// TwinCAT 3 PLC project TXI_SAT
// Title: mr3k3-mr4k3-mr2l1-mr3l1-sat
// Company: SLAC
// ProjectVersion: 0.0.0
// ProgramVersion: 3.1.4022.7
// libraries:
//   lcls-twincat-motion, * (SLAC)
//   Tc2_EtherCAT, * (Beckhoff Automation GmbH)
//   Tc2_Standard, * (Beckhoff Automation GmbH)
//   Tc2_System, * (Beckhoff Automation GmbH)
//   Tc3_Module, * (Beckhoff Automation GmbH)
// project tree:
//   / PlcTask.TcTTO
//   POUs/ MAIN.TcPOU
// real-time tasks:
//   TASK PlcTask: cycle T#10ms, priority 20, ADS port 350
// motion (NC):
//   TASK NC-Task 1 SAF: cycle T#2ms, priority 4, ADS port 501
//   TASK NC-Task 1 SVB: cycle T#10ms, priority 8, ADS port 511
//   AXIS M3K3 X (id 1)
//     Dynamic: AccelerationMaximum=100, DecelerationMaximum=100, Acceleration=100, Deceleration=100, DelayTime=0.008
//     Velo: Maximum=0.4
//     OtherSettings: AllowMotionCmdToSlave=true
//     encoder EncType=29
//       EncPara: ScaleFactorNumerator=5e-06, MaxCount=#xffffffff
//         Inc: RefSoftSyncMask=#x0000ffff
//     drive DrvType=24
//       DrvPara: Inverse=true
//         Analog: VeloReferenz=20, ScaleFactorActTorque=0.1
//         TimeComp: TaskDelayCycles=1
//     controller CtrType=2
//       CtrPara: PriorControlFactor=1
//         PosDiffControl: Range=0.3
//         PID: DeadBandPosition=0.1
//         Observer: BandWidth=20
//   AXIS M3K3 Y (id 2)
//     Dynamic: AccelerationMaximum=100, DecelerationMaximum=100, Acceleration=100, Deceleration=100, DelayTime=0.008
//     Velo: Maximum=0.3
//     OtherSettings: AllowMotionCmdToSlave=true
//     encoder EncType=29
//       EncPara: ScaleFactorNumerator=5e-06, MaxCount=#xffffffff
//         Inc: RefSoftSyncMask=#x0000ffff
//     drive DrvType=24
//       DrvPara: Inverse=true
//         Analog: VeloReferenz=1.25, ScaleFactorActTorque=0.1
//         TimeComp: TaskDelayCycles=1
//     controller CtrType=2
//       CtrPara: PriorControlFactor=1
//         PosDiffControl: Range=0.3
//         PID: DeadBandPosition=0.1
//         Observer: BandWidth=20
//   AXIS M3K3 rX (id 3)
//     General: UnitName=urad
//     Dynamic: AccelerationMaximum=100, DecelerationMaximum=100, Acceleration=100, Deceleration=100, DelayTime=0.008
//     Velo: Maximum=35
//     OtherSettings: AllowMotionCmdToSlave=true
//     encoder EncType=29
//       EncPara: ScaleFactorNumerator=0.001796, MaxCount=#xffffffff
//         Inc: RefSoftSyncMask=#x0000ffff
//     drive DrvType=24
//       Analog: VeloReferenz=87.7, ScaleFactorActTorque=0.1
//       TimeComp: TaskDelayCycles=1
//     controller CtrType=2
//       CtrPara: PriorControlFactor=1
//         PosDiffControl: Range=10
//         PID: DeadBandPosition=10
//         Observer: BandWidth=20
//   AXIS M4K3 X (id 4)
//     Dynamic: AccelerationMaximum=100, DecelerationMaximum=100, Acceleration=100, Deceleration=100, DelayTime=0.008
//     Velo: Maximum=0.3
//     OtherSettings: AllowMotionCmdToSlave=true
//     encoder EncType=29
//       EncPara: ScaleFactorNumerator=5e-06, MaxCount=#xffffffff
//         Inc: RefSoftSyncMask=#x0000ffff
//     drive DrvType=24
//       Analog: VeloReferenz=20, ScaleFactorActTorque=0.1
//       TimeComp: TaskDelayCycles=1
//     controller CtrType=2
//       CtrPara: PriorControlFactor=1
//         PosDiffControl: Range=0.3
//         PID: DeadBandPosition=0.1
//         Observer: BandWidth=20
//   AXIS M4K3 Y (id 5)
//     Dynamic: AccelerationMaximum=100, DecelerationMaximum=100, Acceleration=100, Deceleration=100, DelayTime=0.008
//     Velo: Maximum=0.3
//     OtherSettings: AllowMotionCmdToSlave=true
//     encoder EncType=29
//       EncPara: ScaleFactorNumerator=5e-06, MaxCount=#xffffffff
//         Inc: RefSoftSyncMask=#x0000ffff
//     drive DrvType=24
//       DrvPara: Inverse=true
//         Analog: VeloReferenz=1.25, ScaleFactorActTorque=0.1
//         TimeComp: TaskDelayCycles=1
//     controller CtrType=2
//       CtrPara: PriorControlFactor=1
//         PosDiffControl: Range=0.3
//         PID: DeadBandPosition=1
//         Observer: BandWidth=20
//   AXIS M4K3 rY (id 6)
//     General: UnitName=urad
//     Dynamic: AccelerationMaximum=100, DecelerationMaximum=100, Acceleration=100, Deceleration=100, DelayTime=0.008
//     Velo: Maximum=35
//     OtherSettings: AllowMotionCmdToSlave=true
//     encoder EncType=29
//       EncPara: ScaleFactorNumerator=0.0025316, MaxCount=#xffffffff
//         Inc: RefSoftSyncMask=#x0000ffff
//     drive DrvType=24
//       Analog: VeloReferenz=125, ScaleFactorActTorque=0.1
//       TimeComp: TaskDelayCycles=1
//     controller CtrType=2
//       CtrPara: PriorControlFactor=1
//         PosDiffControl: Range=10
//         PID: DeadBandPosition=0.1
//         Observer: BandWidth=20
//   AXIS M2L1 X (id 7)
//     Dynamic: AccelerationMaximum=100, DecelerationMaximum=100, Acceleration=100, Deceleration=100, DelayTime=0.008
//     Velo: Maximum=0.4
//     OtherSettings: AllowMotionCmdToSlave=true
//     encoder EncType=29
//       EncPara: ScaleFactorNumerator=5e-06, MaxCount=#xffffffff
//         Inc: RefSoftSyncMask=#x0000ffff
//     drive DrvType=24
//       DrvPara: Inverse=true
//         Analog: VeloReferenz=20, ScaleFactorActTorque=0.1
//         TimeComp: TaskDelayCycles=1
//     controller CtrType=2
//       CtrPara: PriorControlFactor=1
//         PosDiffControl: Range=0.3
//         PID: DeadBandPosition=0.1
//         Observer: BandWidth=20
//   AXIS M2L1 Y (id 8)
//     Dynamic: AccelerationMaximum=100, DecelerationMaximum=100, Acceleration=100, Deceleration=100, DelayTime=0.008
//     Velo: Maximum=0.3
//     OtherSettings: AllowMotionCmdToSlave=true
//     encoder EncType=29
//       EncPara: ScaleFactorNumerator=5e-06, MaxCount=#xffffffff
//         Inc: RefSoftSyncMask=#x0000ffff
//     drive DrvType=24
//       DrvPara: Inverse=true
//         Analog: VeloReferenz=1.25, ScaleFactorActTorque=0.1
//         TimeComp: TaskDelayCycles=1
//     controller CtrType=2
//       CtrPara: PriorControlFactor=1
//         PosDiffControl: Range=0.3
//         PID: DeadBandPosition=0.1
//         Observer: BandWidth=20
//   AXIS M2L1 rX (id 9)
//     General: UnitName=urad
//     Dynamic: AccelerationMaximum=100, DecelerationMaximum=100, Acceleration=100, Deceleration=100, DelayTime=0.008
//     Velo: Maximum=35
//     OtherSettings: AllowMotionCmdToSlave=true
//     encoder EncType=29
//       EncPara: ScaleFactorNumerator=0.001796, MaxCount=#xffffffff
//         Inc: RefSoftSyncMask=#x0000ffff
//     drive DrvType=24
//       Analog: VeloReferenz=87.7, ScaleFactorActTorque=0.1
//       TimeComp: TaskDelayCycles=1
//     controller CtrType=2
//       CtrPara: PriorControlFactor=1
//         PosDiffControl: Range=10
//         PID: DeadBandPosition=10
//         Observer: BandWidth=20
//   AXIS M3L1 X (id 10)
//     Dynamic: AccelerationMaximum=100, DecelerationMaximum=100, Acceleration=100, Deceleration=100, DelayTime=0.008
//     Velo: Maximum=0.3
//     OtherSettings: AllowMotionCmdToSlave=true
//     encoder EncType=29
//       EncPara: ScaleFactorNumerator=5e-06, MaxCount=#xffffffff
//         Inc: RefSoftSyncMask=#x0000ffff
//     drive DrvType=24
//       DrvPara: Inverse=true
//         Analog: VeloReferenz=20, ScaleFactorActTorque=0.1
//         TimeComp: TaskDelayCycles=1
//     controller CtrType=2
//       CtrPara: PriorControlFactor=1
//         PosDiffControl: Range=0.3
//         PID: DeadBandPosition=0.1
//         Observer: BandWidth=20
//   AXIS M3L1 Y (id 11)
//     Dynamic: AccelerationMaximum=100, DecelerationMaximum=100, Acceleration=100, Deceleration=100, DelayTime=0.008
//     Velo: Maximum=0.35
//     OtherSettings: AllowMotionCmdToSlave=true
//     encoder EncType=29
//       EncPara: ScaleFactorNumerator=5e-06, MaxCount=#xffffffff
//         Inc: RefSoftSyncMask=#x0000ffff
//     drive DrvType=24
//       DrvPara: Inverse=true
//         Analog: VeloReferenz=1.25, ScaleFactorActTorque=0.1
//         TimeComp: TaskDelayCycles=1
//     controller CtrType=2
//       CtrPara: PriorControlFactor=1
//         PosDiffControl: Range=0.3
//         PID: DeadBandPosition=1
//         Observer: BandWidth=20
//   AXIS M3L1 rY (id 12)
//     General: UnitName=urad
//     Dynamic: AccelerationMaximum=100, DecelerationMaximum=100, Acceleration=100, Deceleration=100, DelayTime=0.008
//     Velo: Maximum=35
//     OtherSettings: AllowMotionCmdToSlave=true
//     encoder EncType=29
//       EncPara: ScaleFactorNumerator=0.0025316, MaxCount=#xffffffff
//         Inc: RefSoftSyncMask=#x0000ffff
//     drive DrvType=24
//       Analog: VeloReferenz=125, ScaleFactorActTorque=0.1
//       TimeComp: TaskDelayCycles=1
//     controller CtrType=2
//       CtrPara: PriorControlFactor=1
//         PosDiffControl: Range=10
//         PID: PosExtKp=15, DeadBandPosition=0.1
//         Observer: BandWidth=20
//   AXIS MMS-BEND (id 13)
//     Dynamic: AccelerationMaximum=0.6, DecelerationMaximum=0.6, Acceleration=0.6, Deceleration=0.6, Jerk=1.2, DelayTime=0.008
//     Velo: Maximum=0.05
//     OtherSettings: AllowMotionCmdToSlave=true
//     encoder EncType=29
//       EncPara: ScaleFactorNumerator=1e-06, MaxCount=#xffffffff
//         SoftEndMinControl: Range=6.4549
//         SoftEndMaxControl: Range=16.0941
//         Inc: RefSoftSyncMask=#x0000ffff
//     drive DrvType=24
//       DrvPara: Inverse=true
//         Analog: VeloReferenz=0.1, ScaleFactorActTorque=0.1
//         TimeComp: TaskDelayCycles=1
//     controller CtrType=2
//       CtrPara: PriorControlFactor=1
//         PosDiffControl: Range=0.2
//         PID: PosKp=15, PosExtKp=1, DeadBandPosition=0.001
//         Observer: BandWidth=20
// I/O:
//   DEVICE Device 1 (EtherCAT), AmsNetId 172.21.84.181.2.1
//     Term 1 (EK1200) [EK1200-5000 EtherCAT Power supply (2A E-Bus)]
//       Term 24 (EL3052) [EL3052 2Ch. Ana. Input 4-20mA]
//       Term 25 (EL3202-0010) [EL3202-0010 2Ch. Ana. Input PT100 (RTD), High Precision]
//       Term 26 (EL7031) [EL7031 1Ch. Stepper motor output stage (24V, 1.5A)]
//       Term 2 (EK1122) [EK1122 2 port EtherCAT junction]
//         TXI K (EK1100) [EK1100 EtherCAT Coupler (2A E-Bus)]
//           M3K3 XY (EL5042)
//           M3K3 rX M4K3 X (EL5042)
//           M4K3 YrY (EL5042)
//           Term 7 (EL9221-5000) [EL9221-5000 Overcurrent protection 24V DC, 1Ch., max. 10A, adjustable]
//           M3K3 X (EL7041-0052)
//           M3K3 Y  (EL7041-0052)
//           M3K3 rX (EL7041-0052)
//           Term 11 (EL9221-5000)
//           M4K3 X (EL7041-0052)
//           M4K3 Y (EL7041-0052) [EL7041-0052 1Ch. Stepper motor output stage (50V, 5A)]
//           M4K3 rY (EL7041-0052) [EL7041-0052 1Ch. Stepper motor output stage (50V, 5A)]
//           Term 15 (EL9410) [EL9410 E-Bus Power Supplier  (Diagnostics)]
//           Term 16 (EL1004)
//           Term 17 (EL3204)
//           Term 18 (EL3204)
//           Term 19 (EL3202-0010)
//           Term 20 (EL3202-0010)
//           Term 21 (EL3054)
//           Term 97 (EL9011)
//         Term 22 (EK1100) [EK1100 EtherCAT Coupler (2A E-Bus)]
//           EL7041_MMS_BEND
//           EL5042_MMS_BEND [EL5042 2Ch. BiSS-C Encoder]
//           EL3202-0010_MMS_BEND [EL3202-0010 2Ch. Ana. Input PT100 (RTD), High Precision]
//           EL3202-0010_MMS_BEND_2 [EL3202-0010 2Ch. Ana. Input PT100 (RTD), High Precision]
//           Term 30 (EL9011)
//         TXI L (EK1100) [EK1100 EtherCAT Coupler (2A E-Bus)]
//           M2L1 XY (EL5042)
//           M2L1 rX M3L1 X (EL5042)
//           M3L1 YrY(EL5042)
//           Term 48 (EL9221-5000)
//           M2L1 X (EL7041-0052) [EL7041-0052 1Ch. Stepper motor output stage (50V, 5A)]
//           M2L1 Y (EL7041-0052) [EL7041-0052 1Ch. Stepper motor output stage (50V, 5A)]
//           M2L1 rX (EL7041-0052) [EL7041-0052 1Ch. Stepper motor output stage (50V, 5A)]
//           Term 52 (EL9221-5000)
//           M3L1 X (EL7041-0052) [EL7041-0052 1Ch. Stepper motor output stage (50V, 5A)]
//           M3L1 Y (EL7041-0052)
//           M3L1 rY (EL7041-0052) [EL7041-0052 1Ch. Stepper motor output stage (50V, 5A)]
//           Term 56 (EL9410)
//           Term 57 (EL3204)
//           Term 58 (EL3204)
//           Term 59 (EL3202-0010)
//           Term 60 (EL3202-0010)
//           Term 61 (EL3054) [EL3054 4Ch. Ana. Input 4-20mA]
//           Term 63 (EL9011)
// variable links:
//   (this object) <-> Device 1 (EtherCAT)/Term 1 (EK1200)/Term 2 (EK1122)/TXI K (EK1100)/M3K3 X (EL7041-0052)
//     Drive/Inputs/In/nState1 @bit 3 <-> STM Status/Status/Error
//     Drive/Inputs/In/nState1 @bit 5 <-> STM Status/Status/Moving negative
//     Drive/Inputs/In/nState1 @bit 4 <-> STM Status/Status/Moving positive
//     Drive/Inputs/In/nState1 @bit 1 <-> STM Status/Status/Ready
//     Drive/Inputs/In/nState1 <-> STM Status/Status/Ready to enable
//     Drive/Inputs/In/nState1 @bit 6 <-> STM Status/Status/Torque reduced
//     Drive/Inputs/In/nState1 @bit 2 <-> STM Status/Status/Warning
//     Drive/Inputs/In/nState2 @bit 3 <-> STM Status/Status/Digital input 1
//     Drive/Inputs/In/nState2 @bit 4 <-> STM Status/Status/Digital input 2
//     Drive/Inputs/In/nState2 @bit 5 <-> STM Status/Status/Sync error
//     Drive/Inputs/In/nState2 @bit 7 <-> STM Status/Status/TxPDO Toggle
//     Drive/Inputs/In/nState4 @bit 1 <-> WcState/InputToggle
//     Drive/Inputs/In/nState4 <-> WcState/WcState
//     Drive/Outputs/Out/nCtrl1 <-> STM Control/Control/Enable
//     Drive/Outputs/Out/nCtrl1 @bit 2 <-> STM Control/Control/Reduce torque
//     Drive/Outputs/Out/nCtrl1 @bit 1 <-> STM Control/Control/Reset
//     Drive/Outputs/Out/nDataOut2[0] <-> STM Velocity/Velocity
//   (this object) <-> Device 1 (EtherCAT)/Term 1 (EK1200)/Term 2 (EK1122)/TXI K (EK1100)/M3K3 XY (EL5042)
//     Enc/Inputs/In/nComState @bit 1 <-> WcState/InputToggle
//     Enc/Inputs/In/nComState <-> WcState/WcState
//     Enc/Inputs/In/nDataIn1 <-> FB Inputs Channel 1/Position
//     Enc/Inputs/In/nDataIn1 <-> FB Inputs Channel 2/Position
//     Enc/Inputs/In/nState1 @bit 12 <-> FB Inputs Channel 1/Status/Diag
//     Enc/Inputs/In/nState1 @bit 12 <-> FB Inputs Channel 2/Status/Diag
//     Enc/Inputs/In/nState1 @bit 1 <-> FB Inputs Channel 1/Status/Error
//     Enc/Inputs/In/nState1 @bit 1 <-> FB Inputs Channel 2/Status/Error
//     Enc/Inputs/In/nState1 @bit 14 <-> FB Inputs Channel 1/Status/Input cycle counter
//     Enc/Inputs/In/nState1 @bit 14 <-> FB Inputs Channel 2/Status/Input cycle counter
//     Enc/Inputs/In/nState1 @bit 2 <-> FB Inputs Channel 1/Status/Ready
//     Enc/Inputs/In/nState1 @bit 2 <-> FB Inputs Channel 2/Status/Ready
//     Enc/Inputs/In/nState1 @bit 13 <-> FB Inputs Channel 1/Status/TxPDO State
//     Enc/Inputs/In/nState1 @bit 13 <-> FB Inputs Channel 2/Status/TxPDO State
//     Enc/Inputs/In/nState1 <-> FB Inputs Channel 1/Status/Warning
//     Enc/Inputs/In/nState1 <-> FB Inputs Channel 2/Status/Warning
//   (this object) <-> Device 1 (EtherCAT)/Term 1 (EK1200)/Term 2 (EK1122)/TXI K (EK1100)/M3K3 Y  (EL7041-0052)
//     Drive/Inputs/In/nState1 @bit 3 <-> STM Status/Status/Error
//     Drive/Inputs/In/nState1 @bit 5 <-> STM Status/Status/Moving negative
//     Drive/Inputs/In/nState1 @bit 4 <-> STM Status/Status/Moving positive
//     Drive/Inputs/In/nState1 @bit 1 <-> STM Status/Status/Ready
//     Drive/Inputs/In/nState1 <-> STM Status/Status/Ready to enable
//     Drive/Inputs/In/nState1 @bit 6 <-> STM Status/Status/Torque reduced
//     Drive/Inputs/In/nState1 @bit 2 <-> STM Status/Status/Warning
//     Drive/Inputs/In/nState2 @bit 5 <-> STM Status/Status/Sync error
//     Drive/Inputs/In/nState2 @bit 7 <-> STM Status/Status/TxPDO Toggle
//     Drive/Inputs/In/nState4 @bit 1 <-> WcState/InputToggle
//     Drive/Inputs/In/nState4 <-> WcState/WcState
//     Drive/Outputs/Out/nCtrl1 <-> STM Control/Control/Enable
//     Drive/Outputs/Out/nCtrl1 @bit 2 <-> STM Control/Control/Reduce torque
//     Drive/Outputs/Out/nCtrl1 @bit 1 <-> STM Control/Control/Reset
//     Drive/Outputs/Out/nDataOut2[0] <-> STM Velocity/Velocity
//   (this object) <-> Device 1 (EtherCAT)/Term 1 (EK1200)/Term 2 (EK1122)/TXI K (EK1100)/M3K3 rX (EL7041-0052)
//     Drive/Inputs/In/nState1 @bit 3 <-> STM Status/Status/Error
//     Drive/Inputs/In/nState1 @bit 5 <-> STM Status/Status/Moving negative
//     Drive/Inputs/In/nState1 @bit 4 <-> STM Status/Status/Moving positive
//     Drive/Inputs/In/nState1 @bit 1 <-> STM Status/Status/Ready
//     Drive/Inputs/In/nState1 <-> STM Status/Status/Ready to enable
//     Drive/Inputs/In/nState1 @bit 6 <-> STM Status/Status/Torque reduced
//     Drive/Inputs/In/nState1 @bit 2 <-> STM Status/Status/Warning
//     Drive/Inputs/In/nState2 @bit 3 <-> STM Status/Status/Digital input 1
//     Drive/Inputs/In/nState2 @bit 4 <-> STM Status/Status/Digital input 2
//     Drive/Inputs/In/nState2 @bit 5 <-> STM Status/Status/Sync error
//     Drive/Inputs/In/nState2 @bit 7 <-> STM Status/Status/TxPDO Toggle
//     Drive/Inputs/In/nState4 @bit 1 <-> WcState/InputToggle
//     Drive/Inputs/In/nState4 <-> WcState/WcState
//     Drive/Outputs/Out/nCtrl1 <-> STM Control/Control/Enable
//     Drive/Outputs/Out/nCtrl1 @bit 2 <-> STM Control/Control/Reduce torque
//     Drive/Outputs/Out/nCtrl1 @bit 1 <-> STM Control/Control/Reset
//     Drive/Outputs/Out/nDataOut2[0] <-> STM Velocity/Velocity
//   (this object) <-> Device 1 (EtherCAT)/Term 1 (EK1200)/Term 2 (EK1122)/TXI K (EK1100)/M3K3 rX M4K3 X (EL5042)
//     Enc/Inputs/In/nComState @bit 1 <-> WcState/InputToggle
//     Enc/Inputs/In/nComState <-> WcState/WcState
//     Enc/Inputs/In/nDataIn1 <-> FB Inputs Channel 1/Position
//     Enc/Inputs/In/nDataIn1 <-> FB Inputs Channel 2/Position
//     Enc/Inputs/In/nState1 @bit 12 <-> FB Inputs Channel 1/Status/Diag
//     Enc/Inputs/In/nState1 @bit 12 <-> FB Inputs Channel 2/Status/Diag
//     Enc/Inputs/In/nState1 @bit 1 <-> FB Inputs Channel 1/Status/Error
//     Enc/Inputs/In/nState1 @bit 1 <-> FB Inputs Channel 2/Status/Error
//     Enc/Inputs/In/nState1 @bit 14 <-> FB Inputs Channel 1/Status/Input cycle counter
//     Enc/Inputs/In/nState1 @bit 14 <-> FB Inputs Channel 2/Status/Input cycle counter
//     Enc/Inputs/In/nState1 @bit 2 <-> FB Inputs Channel 1/Status/Ready
//     Enc/Inputs/In/nState1 @bit 2 <-> FB Inputs Channel 2/Status/Ready
//     Enc/Inputs/In/nState1 @bit 13 <-> FB Inputs Channel 1/Status/TxPDO State
//     Enc/Inputs/In/nState1 @bit 13 <-> FB Inputs Channel 2/Status/TxPDO State
//     Enc/Inputs/In/nState1 <-> FB Inputs Channel 1/Status/Warning
//     Enc/Inputs/In/nState1 <-> FB Inputs Channel 2/Status/Warning
//   (this object) <-> Device 1 (EtherCAT)/Term 1 (EK1200)/Term 2 (EK1122)/TXI K (EK1100)/M4K3 X (EL7041-0052)
//     Drive/Inputs/In/nState1 @bit 3 <-> STM Status/Status/Error
//     Drive/Inputs/In/nState1 @bit 5 <-> STM Status/Status/Moving negative
//     Drive/Inputs/In/nState1 @bit 4 <-> STM Status/Status/Moving positive
//     Drive/Inputs/In/nState1 @bit 1 <-> STM Status/Status/Ready
//     Drive/Inputs/In/nState1 <-> STM Status/Status/Ready to enable
//     Drive/Inputs/In/nState1 @bit 6 <-> STM Status/Status/Torque reduced
//     Drive/Inputs/In/nState1 @bit 2 <-> STM Status/Status/Warning
//     Drive/Inputs/In/nState2 @bit 5 <-> STM Status/Status/Sync error
//     Drive/Inputs/In/nState2 @bit 7 <-> STM Status/Status/TxPDO Toggle
//     Drive/Inputs/In/nState4 @bit 1 <-> WcState/InputToggle
//     Drive/Inputs/In/nState4 <-> WcState/WcState
//     Drive/Outputs/Out/nCtrl1 <-> STM Control/Control/Enable
//     Drive/Outputs/Out/nCtrl1 @bit 2 <-> STM Control/Control/Reduce torque
//     Drive/Outputs/Out/nCtrl1 @bit 1 <-> STM Control/Control/Reset
//     Drive/Outputs/Out/nDataOut2[0] <-> STM Velocity/Velocity
//   (this object) <-> Device 1 (EtherCAT)/Term 1 (EK1200)/Term 2 (EK1122)/TXI K (EK1100)/M4K3 Y (EL7041-0052)
//     Drive/Inputs/In/nState1 @bit 3 <-> STM Status/Status/Error
//     Drive/Inputs/In/nState1 @bit 5 <-> STM Status/Status/Moving negative
//     Drive/Inputs/In/nState1 @bit 4 <-> STM Status/Status/Moving positive
//     Drive/Inputs/In/nState1 @bit 1 <-> STM Status/Status/Ready
//     Drive/Inputs/In/nState1 <-> STM Status/Status/Ready to enable
//     Drive/Inputs/In/nState1 @bit 6 <-> STM Status/Status/Torque reduced
//     Drive/Inputs/In/nState1 @bit 2 <-> STM Status/Status/Warning
//     Drive/Inputs/In/nState2 @bit 3 <-> STM Status/Status/Digital input 1
//     Drive/Inputs/In/nState2 @bit 4 <-> STM Status/Status/Digital input 2
//     Drive/Inputs/In/nState2 @bit 5 <-> STM Status/Status/Sync error
//     Drive/Inputs/In/nState2 @bit 7 <-> STM Status/Status/TxPDO Toggle
//     Drive/Inputs/In/nState4 @bit 1 <-> WcState/InputToggle
//     Drive/Inputs/In/nState4 <-> WcState/WcState
//     Drive/Outputs/Out/nCtrl1 <-> STM Control/Control/Enable
//     Drive/Outputs/Out/nCtrl1 @bit 2 <-> STM Control/Control/Reduce torque
//     Drive/Outputs/Out/nCtrl1 @bit 1 <-> STM Control/Control/Reset
//     Drive/Outputs/Out/nDataOut2[0] <-> STM Velocity/Velocity
//   (this object) <-> Device 1 (EtherCAT)/Term 1 (EK1200)/Term 2 (EK1122)/TXI K (EK1100)/M4K3 YrY (EL5042)
//     Enc/Inputs/In/nComState @bit 1 <-> WcState/InputToggle
//     Enc/Inputs/In/nComState <-> WcState/WcState
//     Enc/Inputs/In/nDataIn1 <-> FB Inputs Channel 1/Position
//     Enc/Inputs/In/nDataIn1 <-> FB Inputs Channel 2/Position
//     Enc/Inputs/In/nState1 @bit 12 <-> FB Inputs Channel 1/Status/Diag
//     Enc/Inputs/In/nState1 @bit 12 <-> FB Inputs Channel 2/Status/Diag
//     Enc/Inputs/In/nState1 @bit 1 <-> FB Inputs Channel 1/Status/Error
//     Enc/Inputs/In/nState1 @bit 1 <-> FB Inputs Channel 2/Status/Error
//     Enc/Inputs/In/nState1 @bit 14 <-> FB Inputs Channel 1/Status/Input cycle counter
//     Enc/Inputs/In/nState1 @bit 14 <-> FB Inputs Channel 2/Status/Input cycle counter
//     Enc/Inputs/In/nState1 @bit 2 <-> FB Inputs Channel 1/Status/Ready
//     Enc/Inputs/In/nState1 @bit 2 <-> FB Inputs Channel 2/Status/Ready
//     Enc/Inputs/In/nState1 @bit 13 <-> FB Inputs Channel 1/Status/TxPDO State
//     Enc/Inputs/In/nState1 @bit 13 <-> FB Inputs Channel 2/Status/TxPDO State
//     Enc/Inputs/In/nState1 <-> FB Inputs Channel 1/Status/Warning
//     Enc/Inputs/In/nState1 <-> FB Inputs Channel 2/Status/Warning
//   (this object) <-> Device 1 (EtherCAT)/Term 1 (EK1200)/Term 2 (EK1122)/TXI K (EK1100)/M4K3 rY (EL7041-0052)
//     Drive/Inputs/In/nState1 @bit 3 <-> STM Status/Status/Error
//     Drive/Inputs/In/nState1 @bit 5 <-> STM Status/Status/Moving negative
//     Drive/Inputs/In/nState1 @bit 4 <-> STM Status/Status/Moving positive
//     Drive/Inputs/In/nState1 @bit 1 <-> STM Status/Status/Ready
//     Drive/Inputs/In/nState1 <-> STM Status/Status/Ready to enable
//     Drive/Inputs/In/nState1 @bit 6 <-> STM Status/Status/Torque reduced
//     Drive/Inputs/In/nState1 @bit 2 <-> STM Status/Status/Warning
//     Drive/Inputs/In/nState2 @bit 3 <-> STM Status/Status/Digital input 1
//     Drive/Inputs/In/nState2 @bit 4 <-> STM Status/Status/Digital input 2
//     Drive/Inputs/In/nState2 @bit 5 <-> STM Status/Status/Sync error
//     Drive/Inputs/In/nState2 @bit 7 <-> STM Status/Status/TxPDO Toggle
//     Drive/Inputs/In/nState4 @bit 1 <-> WcState/InputToggle
//     Drive/Inputs/In/nState4 <-> WcState/WcState
//     Drive/Outputs/Out/nCtrl1 <-> STM Control/Control/Enable
//     Drive/Outputs/Out/nCtrl1 @bit 2 <-> STM Control/Control/Reduce torque
//     Drive/Outputs/Out/nCtrl1 @bit 1 <-> STM Control/Control/Reset
//     Drive/Outputs/Out/nDataOut2[0] <-> STM Velocity/Velocity
//   (this object) <-> Device 1 (EtherCAT)/Term 1 (EK1200)/Term 2 (EK1122)/TXI L (EK1100)/M2L1 X (EL7041-0052)
//     Drive/Inputs/In/nState1 @bit 3 <-> STM Status/Status/Error
//     Drive/Inputs/In/nState1 @bit 5 <-> STM Status/Status/Moving negative
//     Drive/Inputs/In/nState1 @bit 4 <-> STM Status/Status/Moving positive
//     Drive/Inputs/In/nState1 @bit 1 <-> STM Status/Status/Ready
//     Drive/Inputs/In/nState1 <-> STM Status/Status/Ready to enable
//     Drive/Inputs/In/nState1 @bit 6 <-> STM Status/Status/Torque reduced
//     Drive/Inputs/In/nState1 @bit 2 <-> STM Status/Status/Warning
//     Drive/Inputs/In/nState2 @bit 3 <-> STM Status/Status/Digital input 1
//     Drive/Inputs/In/nState2 @bit 4 <-> STM Status/Status/Digital input 2
//     Drive/Inputs/In/nState2 @bit 5 <-> STM Status/Status/Sync error
//     Drive/Inputs/In/nState2 @bit 7 <-> STM Status/Status/TxPDO Toggle
//     Drive/Inputs/In/nState4 @bit 1 <-> WcState/InputToggle
//     Drive/Inputs/In/nState4 <-> WcState/WcState
//     Drive/Outputs/Out/nCtrl1 <-> STM Control/Control/Enable
//     Drive/Outputs/Out/nCtrl1 @bit 2 <-> STM Control/Control/Reduce torque
//     Drive/Outputs/Out/nCtrl1 @bit 1 <-> STM Control/Control/Reset
//     Drive/Outputs/Out/nDataOut2[0] <-> STM Velocity/Velocity
//   (this object) <-> Device 1 (EtherCAT)/Term 1 (EK1200)/Term 2 (EK1122)/TXI L (EK1100)/M2L1 XY (EL5042)
//     Enc/Inputs/In/nComState @bit 1 <-> WcState/InputToggle
//     Enc/Inputs/In/nComState <-> WcState/WcState
//     Enc/Inputs/In/nDataIn1 <-> FB Inputs Channel 1/Position
//     Enc/Inputs/In/nDataIn1 <-> FB Inputs Channel 2/Position
//     Enc/Inputs/In/nState1 @bit 12 <-> FB Inputs Channel 1/Status/Diag
//     Enc/Inputs/In/nState1 @bit 12 <-> FB Inputs Channel 2/Status/Diag
//     Enc/Inputs/In/nState1 @bit 1 <-> FB Inputs Channel 1/Status/Error
//     Enc/Inputs/In/nState1 @bit 1 <-> FB Inputs Channel 2/Status/Error
//     Enc/Inputs/In/nState1 @bit 14 <-> FB Inputs Channel 1/Status/Input cycle counter
//     Enc/Inputs/In/nState1 @bit 14 <-> FB Inputs Channel 2/Status/Input cycle counter
//     Enc/Inputs/In/nState1 @bit 2 <-> FB Inputs Channel 1/Status/Ready
//     Enc/Inputs/In/nState1 @bit 2 <-> FB Inputs Channel 2/Status/Ready
//     Enc/Inputs/In/nState1 @bit 13 <-> FB Inputs Channel 1/Status/TxPDO State
//     Enc/Inputs/In/nState1 @bit 13 <-> FB Inputs Channel 2/Status/TxPDO State
//     Enc/Inputs/In/nState1 <-> FB Inputs Channel 1/Status/Warning
//     Enc/Inputs/In/nState1 <-> FB Inputs Channel 2/Status/Warning
//   (this object) <-> Device 1 (EtherCAT)/Term 1 (EK1200)/Term 2 (EK1122)/TXI L (EK1100)/M2L1 Y (EL7041-0052)
//     Drive/Inputs/In/nState1 @bit 3 <-> STM Status/Status/Error
//     Drive/Inputs/In/nState1 @bit 5 <-> STM Status/Status/Moving negative
//     Drive/Inputs/In/nState1 @bit 4 <-> STM Status/Status/Moving positive
//     Drive/Inputs/In/nState1 @bit 1 <-> STM Status/Status/Ready
//     Drive/Inputs/In/nState1 <-> STM Status/Status/Ready to enable
//     Drive/Inputs/In/nState1 @bit 6 <-> STM Status/Status/Torque reduced
//     Drive/Inputs/In/nState1 @bit 2 <-> STM Status/Status/Warning
//     Drive/Inputs/In/nState2 @bit 3 <-> STM Status/Status/Digital input 1
//     Drive/Inputs/In/nState2 @bit 4 <-> STM Status/Status/Digital input 2
//     Drive/Inputs/In/nState2 @bit 5 <-> STM Status/Status/Sync error
//     Drive/Inputs/In/nState2 @bit 7 <-> STM Status/Status/TxPDO Toggle
//     Drive/Inputs/In/nState4 @bit 1 <-> WcState/InputToggle
//     Drive/Inputs/In/nState4 <-> WcState/WcState
//     Drive/Outputs/Out/nCtrl1 <-> STM Control/Control/Enable
//     Drive/Outputs/Out/nCtrl1 @bit 2 <-> STM Control/Control/Reduce torque
//     Drive/Outputs/Out/nCtrl1 @bit 1 <-> STM Control/Control/Reset
//     Drive/Outputs/Out/nDataOut2[0] <-> STM Velocity/Velocity
//   (this object) <-> Device 1 (EtherCAT)/Term 1 (EK1200)/Term 2 (EK1122)/TXI L (EK1100)/M2L1 rX (EL7041-0052)
//     Drive/Inputs/In/nState1 @bit 3 <-> STM Status/Status/Error
//     Drive/Inputs/In/nState1 @bit 5 <-> STM Status/Status/Moving negative
//     Drive/Inputs/In/nState1 @bit 4 <-> STM Status/Status/Moving positive
//     Drive/Inputs/In/nState1 @bit 1 <-> STM Status/Status/Ready
//     Drive/Inputs/In/nState1 <-> STM Status/Status/Ready to enable
//     Drive/Inputs/In/nState1 @bit 6 <-> STM Status/Status/Torque reduced
//     Drive/Inputs/In/nState1 @bit 2 <-> STM Status/Status/Warning
//     Drive/Inputs/In/nState2 @bit 3 <-> STM Status/Status/Digital input 1
//     Drive/Inputs/In/nState2 @bit 4 <-> STM Status/Status/Digital input 2
//     Drive/Inputs/In/nState2 @bit 5 <-> STM Status/Status/Sync error
//     Drive/Inputs/In/nState2 @bit 7 <-> STM Status/Status/TxPDO Toggle
//     Drive/Inputs/In/nState4 @bit 1 <-> WcState/InputToggle
//     Drive/Inputs/In/nState4 <-> WcState/WcState
//     Drive/Outputs/Out/nCtrl1 <-> STM Control/Control/Enable
//     Drive/Outputs/Out/nCtrl1 @bit 2 <-> STM Control/Control/Reduce torque
//     Drive/Outputs/Out/nCtrl1 @bit 1 <-> STM Control/Control/Reset
//     Drive/Outputs/Out/nDataOut2[0] <-> STM Velocity/Velocity
//   (this object) <-> Device 1 (EtherCAT)/Term 1 (EK1200)/Term 2 (EK1122)/TXI L (EK1100)/M2L1 rX M3L1 X (EL5042)
//     Enc/Inputs/In/nComState @bit 1 <-> WcState/InputToggle
//     Enc/Inputs/In/nComState <-> WcState/WcState
//     Enc/Inputs/In/nDataIn1 <-> FB Inputs Channel 1/Position
//     Enc/Inputs/In/nDataIn1 <-> FB Inputs Channel 2/Position
//     Enc/Inputs/In/nState1 @bit 12 <-> FB Inputs Channel 1/Status/Diag
//     Enc/Inputs/In/nState1 @bit 12 <-> FB Inputs Channel 2/Status/Diag
//     Enc/Inputs/In/nState1 @bit 1 <-> FB Inputs Channel 1/Status/Error
//     Enc/Inputs/In/nState1 @bit 1 <-> FB Inputs Channel 2/Status/Error
//     Enc/Inputs/In/nState1 @bit 14 <-> FB Inputs Channel 1/Status/Input cycle counter
//     Enc/Inputs/In/nState1 @bit 14 <-> FB Inputs Channel 2/Status/Input cycle counter
//     Enc/Inputs/In/nState1 @bit 2 <-> FB Inputs Channel 1/Status/Ready
//     Enc/Inputs/In/nState1 @bit 2 <-> FB Inputs Channel 2/Status/Ready
//     Enc/Inputs/In/nState1 @bit 13 <-> FB Inputs Channel 1/Status/TxPDO State
//     Enc/Inputs/In/nState1 @bit 13 <-> FB Inputs Channel 2/Status/TxPDO State
//     Enc/Inputs/In/nState1 <-> FB Inputs Channel 1/Status/Warning
//     Enc/Inputs/In/nState1 <-> FB Inputs Channel 2/Status/Warning
//   (this object) <-> Device 1 (EtherCAT)/Term 1 (EK1200)/Term 2 (EK1122)/TXI L (EK1100)/M3L1 X (EL7041-0052)
//     Drive/Inputs/In/nState1 @bit 3 <-> STM Status/Status/Error
//     Drive/Inputs/In/nState1 @bit 5 <-> STM Status/Status/Moving negative
//     Drive/Inputs/In/nState1 @bit 4 <-> STM Status/Status/Moving positive
//     Drive/Inputs/In/nState1 @bit 1 <-> STM Status/Status/Ready
//     Drive/Inputs/In/nState1 <-> STM Status/Status/Ready to enable
//     Drive/Inputs/In/nState1 @bit 6 <-> STM Status/Status/Torque reduced
//     Drive/Inputs/In/nState1 @bit 2 <-> STM Status/Status/Warning
//     Drive/Inputs/In/nState2 @bit 3 <-> STM Status/Status/Digital input 1
//     Drive/Inputs/In/nState2 @bit 4 <-> STM Status/Status/Digital input 2
//     Drive/Inputs/In/nState2 @bit 5 <-> STM Status/Status/Sync error
//     Drive/Inputs/In/nState2 @bit 7 <-> STM Status/Status/TxPDO Toggle
//     Drive/Inputs/In/nState4 @bit 1 <-> WcState/InputToggle
//     Drive/Inputs/In/nState4 <-> WcState/WcState
//     Drive/Outputs/Out/nCtrl1 <-> STM Control/Control/Enable
//     Drive/Outputs/Out/nCtrl1 @bit 2 <-> STM Control/Control/Reduce torque
//     Drive/Outputs/Out/nCtrl1 @bit 1 <-> STM Control/Control/Reset
//     Drive/Outputs/Out/nDataOut2[0] <-> STM Velocity/Velocity
//   (this object) <-> Device 1 (EtherCAT)/Term 1 (EK1200)/Term 2 (EK1122)/TXI L (EK1100)/M3L1 Y (EL7041-0052)
//     Drive/Inputs/In/nState1 @bit 3 <-> STM Status/Status/Error
//     Drive/Inputs/In/nState1 @bit 5 <-> STM Status/Status/Moving negative
//     Drive/Inputs/In/nState1 @bit 4 <-> STM Status/Status/Moving positive
//     Drive/Inputs/In/nState1 @bit 1 <-> STM Status/Status/Ready
//     Drive/Inputs/In/nState1 <-> STM Status/Status/Ready to enable
//     Drive/Inputs/In/nState1 @bit 6 <-> STM Status/Status/Torque reduced
//     Drive/Inputs/In/nState1 @bit 2 <-> STM Status/Status/Warning
//     Drive/Inputs/In/nState2 @bit 3 <-> STM Status/Status/Digital input 1
//     Drive/Inputs/In/nState2 @bit 4 <-> STM Status/Status/Digital input 2
//     Drive/Inputs/In/nState2 @bit 5 <-> STM Status/Status/Sync error
//     Drive/Inputs/In/nState2 @bit 7 <-> STM Status/Status/TxPDO Toggle
//     Drive/Inputs/In/nState4 @bit 1 <-> WcState/InputToggle
//     Drive/Inputs/In/nState4 <-> WcState/WcState
//     Drive/Outputs/Out/nCtrl1 <-> STM Control/Control/Enable
//     Drive/Outputs/Out/nCtrl1 @bit 2 <-> STM Control/Control/Reduce torque
//     Drive/Outputs/Out/nCtrl1 @bit 1 <-> STM Control/Control/Reset
//     Drive/Outputs/Out/nDataOut2[0] <-> STM Velocity/Velocity
//   (this object) <-> Device 1 (EtherCAT)/Term 1 (EK1200)/Term 2 (EK1122)/TXI L (EK1100)/M3L1 YrY(EL5042)
//     Enc/Inputs/In/nComState @bit 1 <-> WcState/InputToggle
//     Enc/Inputs/In/nComState <-> WcState/WcState
//     Enc/Inputs/In/nDataIn1 <-> FB Inputs Channel 1/Position
//     Enc/Inputs/In/nDataIn1 <-> FB Inputs Channel 2/Position
//     Enc/Inputs/In/nState1 @bit 12 <-> FB Inputs Channel 1/Status/Diag
//     Enc/Inputs/In/nState1 @bit 12 <-> FB Inputs Channel 2/Status/Diag
//     Enc/Inputs/In/nState1 @bit 1 <-> FB Inputs Channel 1/Status/Error
//     Enc/Inputs/In/nState1 @bit 1 <-> FB Inputs Channel 2/Status/Error
//     Enc/Inputs/In/nState1 @bit 14 <-> FB Inputs Channel 1/Status/Input cycle counter
//     Enc/Inputs/In/nState1 @bit 14 <-> FB Inputs Channel 2/Status/Input cycle counter
//     Enc/Inputs/In/nState1 @bit 2 <-> FB Inputs Channel 1/Status/Ready
//     Enc/Inputs/In/nState1 @bit 2 <-> FB Inputs Channel 2/Status/Ready
//     Enc/Inputs/In/nState1 @bit 13 <-> FB Inputs Channel 1/Status/TxPDO State
//     Enc/Inputs/In/nState1 @bit 13 <-> FB Inputs Channel 2/Status/TxPDO State
//     Enc/Inputs/In/nState1 <-> FB Inputs Channel 1/Status/Warning
//     Enc/Inputs/In/nState1 <-> FB Inputs Channel 2/Status/Warning
//   (this object) <-> Device 1 (EtherCAT)/Term 1 (EK1200)/Term 2 (EK1122)/TXI L (EK1100)/M3L1 rY (EL7041-0052)
//     Drive/Inputs/In/nState1 @bit 3 <-> STM Status/Status/Error
//     Drive/Inputs/In/nState1 @bit 5 <-> STM Status/Status/Moving negative
//     Drive/Inputs/In/nState1 @bit 4 <-> STM Status/Status/Moving positive
//     Drive/Inputs/In/nState1 @bit 1 <-> STM Status/Status/Ready
//     Drive/Inputs/In/nState1 <-> STM Status/Status/Ready to enable
//     Drive/Inputs/In/nState1 @bit 6 <-> STM Status/Status/Torque reduced
//     Drive/Inputs/In/nState1 @bit 2 <-> STM Status/Status/Warning
//     Drive/Inputs/In/nState2 @bit 3 <-> STM Status/Status/Digital input 1
//     Drive/Inputs/In/nState2 @bit 4 <-> STM Status/Status/Digital input 2
//     Drive/Inputs/In/nState2 @bit 5 <-> STM Status/Status/Sync error
//     Drive/Inputs/In/nState2 @bit 7 <-> STM Status/Status/TxPDO Toggle
//     Drive/Inputs/In/nState4 @bit 1 <-> WcState/InputToggle
//     Drive/Inputs/In/nState4 <-> WcState/WcState
//     Drive/Outputs/Out/nCtrl1 <-> STM Control/Control/Enable
//     Drive/Outputs/Out/nCtrl1 @bit 2 <-> STM Control/Control/Reduce torque
//     Drive/Outputs/Out/nCtrl1 @bit 1 <-> STM Control/Control/Reset
//     Drive/Outputs/Out/nDataOut2[0] <-> STM Velocity/Velocity
//   (this object) <-> Device 1 (EtherCAT)/Term 1 (EK1200)/Term 2 (EK1122)/Term 22 (EK1100)/EL5042_MMS_BEND
//     Enc/Inputs/In/nComState @bit 1 <-> WcState/InputToggle
//     Enc/Inputs/In/nComState <-> WcState/WcState
//     Enc/Inputs/In/nDataIn1 <-> FB Inputs Channel 1/Position
//     Enc/Inputs/In/nState1 @bit 12 <-> FB Inputs Channel 1/Status/Diag
//     Enc/Inputs/In/nState1 @bit 1 <-> FB Inputs Channel 1/Status/Error
//     Enc/Inputs/In/nState1 @bit 14 <-> FB Inputs Channel 1/Status/Input cycle counter
//     Enc/Inputs/In/nState1 @bit 2 <-> FB Inputs Channel 1/Status/Ready
//     Enc/Inputs/In/nState1 @bit 13 <-> FB Inputs Channel 1/Status/TxPDO State
//     Enc/Inputs/In/nState1 <-> FB Inputs Channel 1/Status/Warning
//   (this object) <-> Device 1 (EtherCAT)/Term 1 (EK1200)/Term 2 (EK1122)/Term 22 (EK1100)/EL7041_MMS_BEND
//     Drive/Inputs/In/nState1 @bit 3 <-> STM Status/Status/Error
//     Drive/Inputs/In/nState1 @bit 5 <-> STM Status/Status/Moving negative
//     Drive/Inputs/In/nState1 @bit 4 <-> STM Status/Status/Moving positive
//     Drive/Inputs/In/nState1 @bit 1 <-> STM Status/Status/Ready
//     Drive/Inputs/In/nState1 <-> STM Status/Status/Ready to enable
//     Drive/Inputs/In/nState1 @bit 6 <-> STM Status/Status/Torque reduced
//     Drive/Inputs/In/nState1 @bit 2 <-> STM Status/Status/Warning
//     Drive/Inputs/In/nState2 @bit 3 <-> STM Status/Status/Digital input 1
//     Drive/Inputs/In/nState2 @bit 4 <-> STM Status/Status/Digital input 2
//     Drive/Inputs/In/nState2 @bit 5 <-> STM Status/Status/Sync error
//     Drive/Inputs/In/nState2 @bit 7 <-> STM Status/Status/TxPDO Toggle
//     Drive/Inputs/In/nState4 @bit 1 <-> WcState/InputToggle
//     Drive/Inputs/In/nState4 <-> WcState/WcState
//     Drive/Outputs/Out/nCtrl1 <-> STM Control/Control/Enable
//     Drive/Outputs/Out/nCtrl1 @bit 2 <-> STM Control/Control/Reduce torque
//     Drive/Outputs/Out/nCtrl1 @bit 1 <-> STM Control/Control/Reset
//     Drive/Outputs/Out/nDataOut2[0] <-> STM Velocity/Velocity
//   TXI_SAT Instance <-> Device 1 (EtherCAT)/Term 1 (EK1200)/Term 2 (EK1122)/TXI K (EK1100)/M3K3 X (EL7041-0052)
//     PlcTask Inputs/MAIN.M1.bLimitBackwardEnable <-> STM Status/Status/Digital input 2
//     PlcTask Inputs/MAIN.M1.bLimitForwardEnable <-> STM Status/Status/Digital input 1
//   TXI_SAT Instance <-> Device 1 (EtherCAT)/Term 1 (EK1200)/Term 2 (EK1122)/TXI K (EK1100)/M3K3 XY (EL5042)
//     PlcTask Inputs/MAIN.M1.nRawEncoderULINT <-> FB Inputs Channel 1/Position
//     PlcTask Inputs/MAIN.M2.nRawEncoderULINT <-> FB Inputs Channel 2/Position
//   TXI_SAT Instance <-> Device 1 (EtherCAT)/Term 1 (EK1200)/Term 2 (EK1122)/TXI K (EK1100)/M3K3 Y  (EL7041-0052)
//     PlcTask Inputs/MAIN.M2.bLimitBackwardEnable <-> STM Status/Status/Digital input 2
//     PlcTask Inputs/MAIN.M2.bLimitForwardEnable <-> STM Status/Status/Digital input 1
//   TXI_SAT Instance <-> Device 1 (EtherCAT)/Term 1 (EK1200)/Term 2 (EK1122)/TXI K (EK1100)/M3K3 rX (EL7041-0052)
//     PlcTask Inputs/MAIN.M3.bLimitBackwardEnable <-> STM Status/Status/Digital input 2
//     PlcTask Inputs/MAIN.M3.bLimitForwardEnable <-> STM Status/Status/Digital input 1
//   TXI_SAT Instance <-> Device 1 (EtherCAT)/Term 1 (EK1200)/Term 2 (EK1122)/TXI K (EK1100)/M3K3 rX M4K3 X (EL5042)
//     PlcTask Inputs/MAIN.M3.nRawEncoderULINT <-> FB Inputs Channel 1/Position
//     PlcTask Inputs/MAIN.M4.nRawEncoderULINT <-> FB Inputs Channel 2/Position
//   TXI_SAT Instance <-> Device 1 (EtherCAT)/Term 1 (EK1200)/Term 2 (EK1122)/TXI K (EK1100)/M4K3 X (EL7041-0052)
//     PlcTask Inputs/MAIN.M4.bLimitBackwardEnable <-> STM Status/Status/Digital input 1
//     PlcTask Inputs/MAIN.M4.bLimitForwardEnable <-> STM Status/Status/Digital input 2
//   TXI_SAT Instance <-> Device 1 (EtherCAT)/Term 1 (EK1200)/Term 2 (EK1122)/TXI K (EK1100)/M4K3 Y (EL7041-0052)
//     PlcTask Inputs/MAIN.M5.bLimitBackwardEnable <-> STM Status/Status/Digital input 2
//     PlcTask Inputs/MAIN.M5.bLimitForwardEnable <-> STM Status/Status/Digital input 1
//   TXI_SAT Instance <-> Device 1 (EtherCAT)/Term 1 (EK1200)/Term 2 (EK1122)/TXI K (EK1100)/M4K3 YrY (EL5042)
//     PlcTask Inputs/MAIN.M5.nRawEncoderULINT <-> FB Inputs Channel 1/Position
//     PlcTask Inputs/MAIN.M6.nRawEncoderULINT <-> FB Inputs Channel 2/Position
//   TXI_SAT Instance <-> Device 1 (EtherCAT)/Term 1 (EK1200)/Term 2 (EK1122)/TXI K (EK1100)/M4K3 rY (EL7041-0052)
//     PlcTask Inputs/MAIN.M6.bLimitBackwardEnable <-> STM Status/Status/Digital input 2
//     PlcTask Inputs/MAIN.M6.bLimitForwardEnable <-> STM Status/Status/Digital input 1
//   TXI_SAT Instance <-> Device 1 (EtherCAT)/Term 1 (EK1200)/Term 2 (EK1122)/TXI K (EK1100)/Term 16 (EL1004)
//     PlcTask Inputs/MAIN.bSTOEnable1 <-> Channel 1/Input
//     PlcTask Inputs/MAIN.bSTOEnable2 <-> Channel 2/Input
//   TXI_SAT Instance <-> Device 1 (EtherCAT)/Term 1 (EK1200)/Term 2 (EK1122)/TXI L (EK1100)/M2L1 X (EL7041-0052)
//     PlcTask Inputs/MAIN.M7.bLimitBackwardEnable <-> STM Status/Status/Digital input 2
//     PlcTask Inputs/MAIN.M7.bLimitForwardEnable <-> STM Status/Status/Digital input 1
//   TXI_SAT Instance <-> Device 1 (EtherCAT)/Term 1 (EK1200)/Term 2 (EK1122)/TXI L (EK1100)/M2L1 XY (EL5042)
//     PlcTask Inputs/MAIN.M7.nRawEncoderULINT <-> FB Inputs Channel 1/Position
//     PlcTask Inputs/MAIN.M8.nRawEncoderULINT <-> FB Inputs Channel 2/Position
//   TXI_SAT Instance <-> Device 1 (EtherCAT)/Term 1 (EK1200)/Term 2 (EK1122)/TXI L (EK1100)/M2L1 Y (EL7041-0052)
//     PlcTask Inputs/MAIN.M8.bLimitBackwardEnable <-> STM Status/Status/Digital input 2
//     PlcTask Inputs/MAIN.M8.bLimitForwardEnable <-> STM Status/Status/Digital input 1
//   TXI_SAT Instance <-> Device 1 (EtherCAT)/Term 1 (EK1200)/Term 2 (EK1122)/TXI L (EK1100)/M2L1 rX (EL7041-0052)
//     PlcTask Inputs/MAIN.M9.bLimitBackwardEnable <-> STM Status/Status/Digital input 2
//     PlcTask Inputs/MAIN.M9.bLimitForwardEnable <-> STM Status/Status/Digital input 1
//   TXI_SAT Instance <-> Device 1 (EtherCAT)/Term 1 (EK1200)/Term 2 (EK1122)/TXI L (EK1100)/M2L1 rX M3L1 X (EL5042)
//     PlcTask Inputs/MAIN.M10.nRawEncoderULINT <-> FB Inputs Channel 2/Position
//     PlcTask Inputs/MAIN.M9.nRawEncoderULINT <-> FB Inputs Channel 1/Position
//   TXI_SAT Instance <-> Device 1 (EtherCAT)/Term 1 (EK1200)/Term 2 (EK1122)/TXI L (EK1100)/M3L1 X (EL7041-0052)
//     PlcTask Inputs/MAIN.M10.bLimitBackwardEnable <-> STM Status/Status/Digital input 2
//     PlcTask Inputs/MAIN.M10.bLimitForwardEnable <-> STM Status/Status/Digital input 1
//   TXI_SAT Instance <-> Device 1 (EtherCAT)/Term 1 (EK1200)/Term 2 (EK1122)/TXI L (EK1100)/M3L1 Y (EL7041-0052)
//     PlcTask Inputs/MAIN.M11.bLimitBackwardEnable <-> STM Status/Status/Digital input 2
//     PlcTask Inputs/MAIN.M11.bLimitForwardEnable <-> STM Status/Status/Digital input 1
//   TXI_SAT Instance <-> Device 1 (EtherCAT)/Term 1 (EK1200)/Term 2 (EK1122)/TXI L (EK1100)/M3L1 YrY(EL5042)
//     PlcTask Inputs/MAIN.M11.nRawEncoderULINT <-> FB Inputs Channel 1/Position
//     PlcTask Inputs/MAIN.M12.nRawEncoderULINT <-> FB Inputs Channel 2/Position
//   TXI_SAT Instance <-> Device 1 (EtherCAT)/Term 1 (EK1200)/Term 2 (EK1122)/TXI L (EK1100)/M3L1 rY (EL7041-0052)
//     PlcTask Inputs/MAIN.M12.bLimitBackwardEnable <-> STM Status/Status/Digital input 2
//     PlcTask Inputs/MAIN.M12.bLimitForwardEnable <-> STM Status/Status/Digital input 1
//   TXI_SAT Instance <-> Device 1 (EtherCAT)/Term 1 (EK1200)/Term 2 (EK1122)/Term 22 (EK1100)/EL5042_MMS_BEND
//     PlcTask Inputs/MAIN.M13.nRawEncoderULINT <-> FB Inputs Channel 1/Position
//   TXI_SAT Instance <-> Device 1 (EtherCAT)/Term 1 (EK1200)/Term 2 (EK1122)/Term 22 (EK1100)/EL7041_MMS_BEND
//     PlcTask Inputs/MAIN.M13.bLimitBackwardEnable <-> STM Status/Status/Digital input 2
//     PlcTask Inputs/MAIN.M13.bLimitForwardEnable <-> STM Status/Status/Digital input 1
//   TXI_SAT Instance <-> NC-Task 1 SAF/Axes/M2L1 X
//     PlcTask Inputs/MAIN.M7.Axis.NcToPlc <-> Outputs/ToPlc
//     PlcTask Outputs/MAIN.M7.Axis.PlcToNc <-> Inputs/FromPlc
//   TXI_SAT Instance <-> NC-Task 1 SAF/Axes/M2L1 Y
//     PlcTask Inputs/MAIN.M8.Axis.NcToPlc <-> Outputs/ToPlc
//     PlcTask Outputs/MAIN.M8.Axis.PlcToNc <-> Inputs/FromPlc
//   TXI_SAT Instance <-> NC-Task 1 SAF/Axes/M2L1 rX
//     PlcTask Inputs/MAIN.M9.Axis.NcToPlc <-> Outputs/ToPlc
//     PlcTask Outputs/MAIN.M9.Axis.PlcToNc <-> Inputs/FromPlc
//   TXI_SAT Instance <-> NC-Task 1 SAF/Axes/M3K3 X
//     PlcTask Inputs/MAIN.M1.Axis.NcToPlc <-> Outputs/ToPlc
//     PlcTask Outputs/MAIN.M1.Axis.PlcToNc <-> Inputs/FromPlc
//   TXI_SAT Instance <-> NC-Task 1 SAF/Axes/M3K3 Y
//     PlcTask Inputs/MAIN.M2.Axis.NcToPlc <-> Outputs/ToPlc
//     PlcTask Outputs/MAIN.M2.Axis.PlcToNc <-> Inputs/FromPlc
//   TXI_SAT Instance <-> NC-Task 1 SAF/Axes/M3K3 rX
//     PlcTask Inputs/MAIN.M3.Axis.NcToPlc <-> Outputs/ToPlc
//     PlcTask Outputs/MAIN.M3.Axis.PlcToNc <-> Inputs/FromPlc
//   TXI_SAT Instance <-> NC-Task 1 SAF/Axes/M3L1 X
//     PlcTask Inputs/MAIN.M10.Axis.NcToPlc <-> Outputs/ToPlc
//     PlcTask Outputs/MAIN.M10.Axis.PlcToNc <-> Inputs/FromPlc
//   TXI_SAT Instance <-> NC-Task 1 SAF/Axes/M3L1 Y
//     PlcTask Inputs/MAIN.M11.Axis.NcToPlc <-> Outputs/ToPlc
//     PlcTask Outputs/MAIN.M11.Axis.PlcToNc <-> Inputs/FromPlc
//   TXI_SAT Instance <-> NC-Task 1 SAF/Axes/M3L1 rY
//     PlcTask Inputs/MAIN.M12.Axis.NcToPlc <-> Outputs/ToPlc
//     PlcTask Outputs/MAIN.M12.Axis.PlcToNc <-> Inputs/FromPlc
//   TXI_SAT Instance <-> NC-Task 1 SAF/Axes/M4K3 X
//     PlcTask Inputs/MAIN.M4.Axis.NcToPlc <-> Outputs/ToPlc
//     PlcTask Outputs/MAIN.M4.Axis.PlcToNc <-> Inputs/FromPlc
//   TXI_SAT Instance <-> NC-Task 1 SAF/Axes/M4K3 Y
//     PlcTask Inputs/MAIN.M5.Axis.NcToPlc <-> Outputs/ToPlc
//     PlcTask Outputs/MAIN.M5.Axis.PlcToNc <-> Inputs/FromPlc
//   TXI_SAT Instance <-> NC-Task 1 SAF/Axes/M4K3 rY
//     PlcTask Inputs/MAIN.M6.Axis.NcToPlc <-> Outputs/ToPlc
//     PlcTask Outputs/MAIN.M6.Axis.PlcToNc <-> Inputs/FromPlc
//   TXI_SAT Instance <-> NC-Task 1 SAF/Axes/MMS-BEND
//     PlcTask Inputs/MAIN.M13.Axis.NcToPlc <-> Outputs/ToPlc
//     PlcTask Outputs/MAIN.M13.Axis.PlcToNc <-> Inputs/FromPlc

CONFIGURATION TXI_SAT
    RESOURCE PLC ON TwinCAT3
        TASK PlcTask(INTERVAL := T#10ms, PRIORITY := 20);
        PROGRAM MAIN WITH PlcTask : MAIN;
    END_RESOURCE
END_CONFIGURATION

// ---- POUs/MAIN.TcPOU
PROGRAM MAIN
VAR
	{attribute 'TcLinkTo' := '.bLimitForwardEnable:=TIIB[M3K3 X (EL7041-0052)]^STM Status^Status^Digital input 1;
                              .bLimitBackwardEnable:=TIIB[M3K3 X (EL7041-0052)]^STM Status^Status^Digital input 2;
                              .nRawEncoderULINT:=TIIB[M3K3 XY (EL5042)]^FB Inputs Channel 1^Position'}
	{attribute 'pytmc' := '
			pv: MR3K3:KBV:MMS:X
	'}
	 M1 : DUT_MotionStage := (nEnableMode:=ENUM_StageEnableMode.ALWAYS, bPowerSelf:=TRUE);
    fbMotionStageM1 : FB_MotionStage;
	
	{attribute 'TcLinkTo' := '.bLimitForwardEnable:=TIIB[M3K3 Y (EL7041-0052)]^STM Status^Status^Digital input 1;
                              .bLimitBackwardEnable:=TIIB[M3K3 Y (EL7041-0052)]^STM Status^Status^Digital input 2;
                              .nRawEncoderULINT:=TIIB[M3K3 XY (EL5042)]^FB Inputs Channel 2^Position'}
	{attribute 'pytmc' := '
			pv: MR3K3:KBV:MMS:Y
	'}
	 M2 : DUT_MotionStage := (nEnableMode:=ENUM_StageEnableMode.ALWAYS, bPowerSelf:=TRUE);
    fbMotionStageM2 : FB_MotionStage;
	{attribute 'TcLinkTo' := '.bLimitForwardEnable:=TIIB[M3K3 rX (EL7041-0052)]^STM Status^Status^Digital input 1;
                              .bLimitBackwardEnable:=TIIB[M3K3 rX (EL7041-0052)]^STM Status^Status^Digital input 2;
                              .nRawEncoderULINT:=TIIB[M3K3 rX M4K3 X (EL5042)]^FB Inputs Channel 1^Position'}
	{attribute 'pytmc' := '
			pv: MR3K3:KBV:MMS:PITCH
	'}
// theta x
	 M3 : DUT_MotionStage := (nEnableMode:=ENUM_StageEnableMode.ALWAYS, bPowerSelf:=TRUE);
    fbMotionStageM3 : FB_MotionStage;
	
	{attribute 'TcLinkTo' := '.bLimitForwardEnable:=TIIB[M4K3 X (EL7041-0052)]^STM Status^Status^Digital input 2;
                              .bLimitBackwardEnable:=TIIB[M4K3 X (EL7041-0052)]^STM Status^Status^Digital input 1;
                              .nRawEncoderULINT:=TIIB[M3K3 rX M4K3 X (EL5042)]^FB Inputs Channel 2^Position'}
	{attribute 'pytmc' := '
			pv: MR4K3:KBH:MMS:X
	'}
	 M4 : DUT_MotionStage := (nEnableMode:=ENUM_StageEnableMode.ALWAYS, bPowerSelf:=TRUE);
    fbMotionStageM4 : FB_MotionStage;
	 
	{attribute 'TcLinkTo' := '.bLimitForwardEnable:=TIIB[M4K3 Y (EL7041-0052)]^STM Status^Status^Digital input 1;
                              .bLimitBackwardEnable:=TIIB[M4K3 Y (EL7041-0052)]^STM Status^Status^Digital input 2;
                              .nRawEncoderULINT:=TIIB[M4K3 YrY (EL5042)]^FB Inputs Channel 1^Position'}
	{attribute 'pytmc' := '
			pv: MR4K3:KBH:MMS:Y
	'}
	 M5 : DUT_MotionStage := (nEnableMode:=ENUM_StageEnableMode.ALWAYS, bPowerSelf:=TRUE);
    fbMotionStageM5 : FB_MotionStage;
	{attribute 'TcLinkTo' := '.bLimitForwardEnable:=TIIB[M4K3 rY (EL7041-0052)]^STM Status^Status^Digital input 1;
                              .bLimitBackwardEnable:=TIIB[M4K3 rY (EL7041-0052)]^STM Status^Status^Digital input 2;
                              .nRawEncoderULINT:=TIIB[M4K3 YrY (EL5042)]^FB Inputs Channel 2^Position'}
	{attribute 'pytmc' := '
			pv: MR4K3:KBH:MMS:PITCH
	'}
// theta y
     M6 : DUT_MotionStage := (nEnableMode:=ENUM_StageEnableMode.ALWAYS, bPowerSelf:=TRUE);
    fbMotionStageM6 : FB_MotionStage;
    {attribute 'TcLinkTo' := '.bLimitForwardEnable:=TIIB[M2L1 X (EL7041-0052)]^STM Status^Status^Digital input 1;
                              .bLimitBackwardEnable:=TIIB[M2L1 X (EL7041-0052)]^STM Status^Status^Digital input 2;
                              .nRawEncoderULINT:=TIIB[M2L1 XY (EL5042)]^FB Inputs Channel 1^Position'}
	{attribute 'pytmc' := '
			pv: MR2L1:KBV:MMS:X
	'}
	 M7 : DUT_MotionStage := (nEnableMode:=ENUM_StageEnableMode.ALWAYS, bPowerSelf:=TRUE);
    fbMotionStageM7 : FB_MotionStage;
	
	{attribute 'TcLinkTo' := '.bLimitForwardEnable:=TIIB[M2L1 Y (EL7041-0052)]^STM Status^Status^Digital input 1;
                              .bLimitBackwardEnable:=TIIB[M2L1 Y (EL7041-0052)]^STM Status^Status^Digital input 2;
                              .nRawEncoderULINT:=TIIB[M2L1 XY (EL5042)]^FB Inputs Channel 2^Position'}
	{attribute 'pytmc' := '
			pv: MR2L1:KBV:MMS:Y
	'}
	 M8 : DUT_MotionStage := (nEnableMode:=ENUM_StageEnableMode.ALWAYS, bPowerSelf:=TRUE);
    fbMotionStageM8 : FB_MotionStage;
	{attribute 'TcLinkTo' := '.bLimitForwardEnable:=TIIB[M2L1 rX (EL7041-0052)]^STM Status^Status^Digital input 1;
                              .bLimitBackwardEnable:=TIIB[M2L1 rX (EL7041-0052)]^STM Status^Status^Digital input 2;
                              .nRawEncoderULINT:=TIIB[M2L1 rX M3L1 X (EL5042)]^FB Inputs Channel 1^Position'}
	{attribute 'pytmc' := '
			pv: MR2L1:KBV:MMS:PITCH
	'}
// theta x
	 M9 : DUT_MotionStage := (nEnableMode:=ENUM_StageEnableMode.ALWAYS, bPowerSelf:=TRUE);
    fbMotionStageM9 : FB_MotionStage;
	
	{attribute 'TcLinkTo' := '.bLimitForwardEnable:=TIIB[M3L1 X (EL7041-0052)]^STM Status^Status^Digital input 1;
                              .bLimitBackwardEnable:=TIIB[M3L1 X (EL7041-0052)]^STM Status^Status^Digital input 2;
                              .nRawEncoderULINT:=TIIB[M2L1 rX M3L1 X (EL5042)]^FB Inputs Channel 2^Position'}
	{attribute 'pytmc' := '
			pv: MR3L1:KBH:MMS:X
	'}
	 M10 : DUT_MotionStage := (nEnableMode:=ENUM_StageEnableMode.ALWAYS, bPowerSelf:=TRUE);
    fbMotionStageM10 : FB_MotionStage;
	 
	{attribute 'TcLinkTo' := '.bLimitForwardEnable:=TIIB[M3L1 Y (EL7041-0052)]^STM Status^Status^Digital input 1;
                              .bLimitBackwardEnable:=TIIB[M3L1 Y (EL7041-0052)]^STM Status^Status^Digital input 2;
                              .nRawEncoderULINT:=TIIB[M3L1 YrY(EL5042)]^FB Inputs Channel 1^Position'}
	{attribute 'pytmc' := '
			pv: MR3L1:KBH:MMS:Y
	'}
	 M11 : DUT_MotionStage := (nEnableMode:=ENUM_StageEnableMode.ALWAYS, bPowerSelf:=TRUE);
    fbMotionStageM11 : FB_MotionStage;
	{attribute 'TcLinkTo' := '.bLimitForwardEnable:=TIIB[M3L1 rY (EL7041-0052)]^STM Status^Status^Digital input 1;
                              .bLimitBackwardEnable:=TIIB[M3L1 rY (EL7041-0052)]^STM Status^Status^Digital input 2;
                              .nRawEncoderULINT:=TIIB[M3L1 YrY(EL5042)]^FB Inputs Channel 2^Position'}
	{attribute 'pytmc' := '
			pv: MR3L1:KBH:MMS:PITCH
	'}
// theta Y
     M12 : DUT_MotionStage := (nEnableMode:=ENUM_StageEnableMode.ALWAYS, bPowerSelf:=TRUE);
    fbMotionStageM12 : FB_MotionStage;
    //MMMS BEND
        {attribute 'TcLinkTo' := '.bLimitForwardEnable :=TIIB[EL7041_MMS_BEND]^STM Status^Status^Digital input 1;
                                  .bLimitBackwardEnable:=TIIB[EL7041_MMS_BEND]^STM Status^Status^Digital input 2;
                                  .nRawEncoderULINT    := TIIB[EL5042_MMS_BEND]^FB Inputs Channel 1^Position'}
        {attribute 'pytmc' := '
        pv: MMS:BEND:TEST
        '}
        M13 : ST_MotionStage := (nEnableMode:=ENUM_StageEnableMode.ALWAYS, bPowerSelf:=TRUE);
        fbMotionStageM13 : FB_MotionStage;
    {attribute 'TcLinkTo' := 'TIIB[Term 16 (EL1004)]^Channel 1^Input'}
    bSTOEnable1 AT %I* : BOOL;
	
	{attribute 'TcLinkTo' := 'TIIB[Term 16 (EL1004)]^Channel 2^Input'}
    bSTOEnable2 AT %I* : BOOL;
END_VAR

M1.bHardwareEnable := bSTOEnable2 and bSTOEnable1;
M2.bHardwareEnable := bSTOEnable2 and bSTOEnable1;
M3.bHardwareEnable := bSTOEnable2 and bSTOEnable1;
M4.bHardwareEnable := bSTOEnable2 and bSTOEnable1;
M5.bHardwareEnable := bSTOEnable2 and bSTOEnable1;
M6.bHardwareEnable := bSTOEnable2 and bSTOEnable1;

M7.bHardwareEnable := bSTOEnable2 and bSTOEnable1;
M8.bHardwareEnable := bSTOEnable2 and bSTOEnable1;
M9.bHardwareEnable := bSTOEnable2 and bSTOEnable1;
M10.bHardwareEnable := bSTOEnable2 and bSTOEnable1;
M11.bHardwareEnable := bSTOEnable2 and bSTOEnable1;
M12.bHardwareEnable := bSTOEnable2 and bSTOEnable1;
M13.bHardwareEnable := bSTOEnable2 and bSTOEnable1;

fbMotionStageM1(stMotionStage:=M1);
fbMotionStageM2(stMotionStage:=M2);
fbMotionStageM3(stMotionStage:=M3);
fbMotionStageM4(stMotionStage:=M4);
fbMotionStageM5(stMotionStage:=M5);
fbMotionStageM6(stMotionStage:=M6);

fbMotionStageM7(stMotionStage:=M7);
fbMotionStageM8(stMotionStage:=M8);
fbMotionStageM9(stMotionStage:=M9);
fbMotionStageM10(stMotionStage:=M10);
fbMotionStageM11(stMotionStage:=M11);
fbMotionStageM12(stMotionStage:=M12);
fbMotionStageM13(stMotionStage:=M13);

END_PROGRAM
